// TIA Portal V18 export
FUNCTION_BLOCK "Aux_Functions"   // FB16, LAD
TITLE = Aux_Functions
{ S7_Optimized_Access := 'TRUE' }
// Written BY Kristopher Gimenez January 26,2023
// This block is used to control TD auxilarry functions
// stored: AutoNumber false, MemoryReserve 100, SetENOAutomatically false
   VAR
      PTO_Pulse { S7_SetPoint := 'True'} : TP_TIME;
      BUWOpenCLKTOffTime { S7_SetPoint := 'True'} : TP_TIME;
      BUWOpenCLKOnTime { S7_SetPoint := 'True'} : TP_TIME;
      BUWCloseHoldTOF { S7_SetPoint := 'True'} : TOF_TIME;
      MUDoneTP { S7_SetPoint := 'True'} : TP_TIME;
      BUWOpPulse { S7_SetPoint := 'True'} : TP_TIME;
      ElevCl_TON { S7_SetPoint := 'True'} : TON_TIME;
      ElevOpTime_TP { S7_SetPoint := 'True'} : TP_TIME;
      MSVOp_TON { S7_SetPoint := 'True'} : TON_TIME;
      MPRunning_TOF { S7_SetPoint := 'True'} : TOF_TIME;
      MSVCl_TON { S7_SetPoint := 'True'} : TON_TIME;
      BUWMainCl_Int { S7_SetPoint := 'True'} : Bool;
      TDModeMUTrig : Bool;
      TDModeBOTrig { ExternalAccessible := 'False'; ExternalVisible := 'False'; ExternalWritable := 'False'} : Bool;
      ElevOpOnTime : Bool;   // Bool that will be high for 8 seconds while elevator opens
      LinksDisable : Bool;   // Link Tilt Extend and Retract disabled
      ElevClDisable : Bool;   // Disable Close after output on for set time
      MSVClDisable { S7_SetPoint := 'True'} : Bool;   // MSV close disabled due to mud Pump running if high
      MSVOpDisable { S7_SetPoint := 'True'} : Bool;   // Disable after output on for set time
      ElevOpSwTrig : Bool;
      ElevCl_TON_1 { S7_SetPoint := 'True'} : TON_TIME;
      ElevCl_TON_5s { S7_SetPoint := 'True'} : TON_TIME;
   END_VAR
   // PTO_Pulse.PT := T#5s;
   VAR_TEMP   // added for the SCL form of the ladder/FBD networks
      _w1 : Bool;
      _w2 : Bool;
   END_VAR
BEGIN

REGION Network 1: PTO Pulse
   // When PTO is pressed there will be a 5 seconds pulse allowing operations.
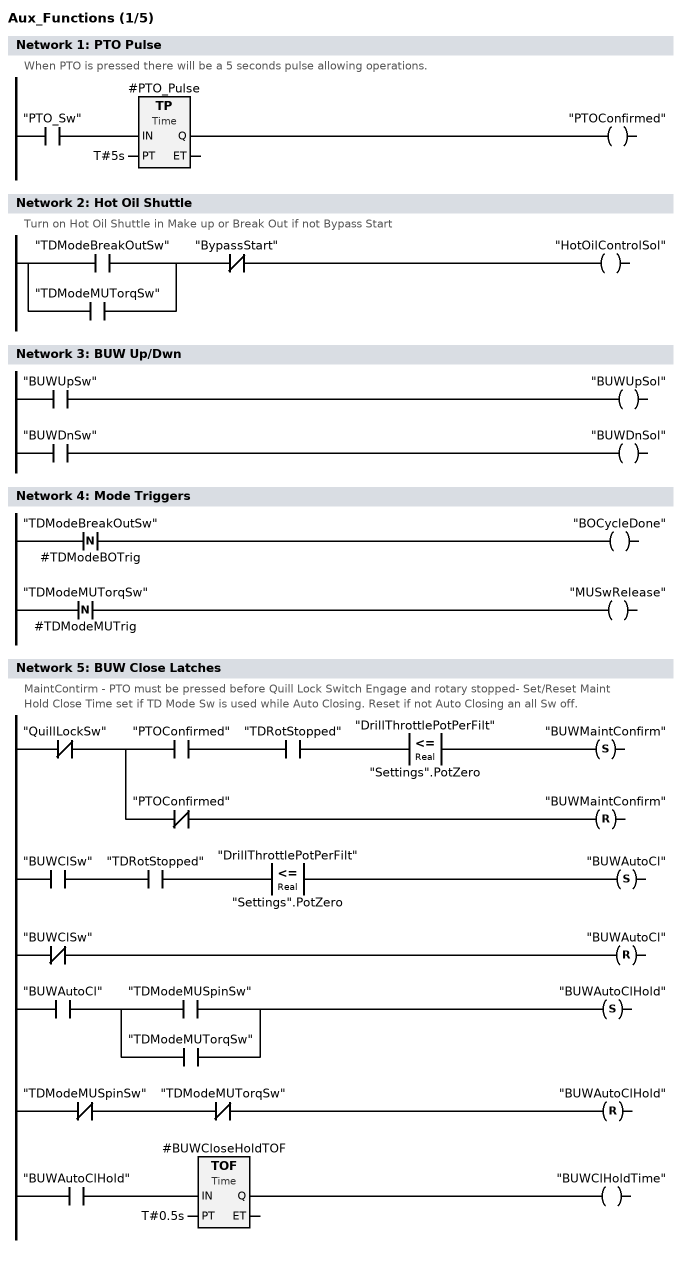
   RUNG wire#powerrail
      Contact( "PTO_Sw" )
      { S7_Templates := "time_type := Time" } #PTO_Pulse.TP(pt := T#5s, et =>)
      Coil( "PTOConfirmed" )
   END_RUNG
   // the same network as SCL:
   #PTO_Pulse(IN := "PTO_Sw", PT := T#5s);   // TP
   "PTOConfirmed" := #PTO_Pulse.Q;
END_REGION

REGION Network 2: Hot Oil Shuttle
   // Turn on Hot Oil Shuttle in Make up or Break Out if not Bypass Start
   RUNG wire#powerrail
      Contact( "TDModeBreakOutSw" )
      wire#w1
      I_Contact( "BypassStart" )
      Coil( "HotOilControlSol" )
   END_RUNG
   RUNG wire#powerrail
      Contact( "TDModeMUTorqSw" )
   END_RUNG wire#w1
   // the same network as SCL:
   "HotOilControlSol" := ("TDModeBreakOutSw" OR "TDModeMUTorqSw") AND NOT "BypassStart";
END_REGION

REGION Network 3: BUW Up/Dwn
   RUNG wire#powerrail
      Contact( "BUWUpSw" )
      Coil( "BUWUpSol" )
   END_RUNG
   RUNG wire#powerrail
      Contact( "BUWDnSw" )
      Coil( "BUWDnSol" )
   END_RUNG
   // the same network as SCL:
   "BUWUpSol" := "BUWUpSw";
   "BUWDnSol" := "BUWDnSw";
END_REGION

REGION Network 4: Mode Triggers
   RUNG wire#powerrail
      N_Contact(operand := "TDModeBreakOutSw", bit := #TDModeBOTrig)
      Coil( "BOCycleDone" )
   END_RUNG
   RUNG wire#powerrail
      N_Contact(operand := "TDModeMUTorqSw", bit := #TDModeMUTrig)
      Coil( "MUSwRelease" )
   END_RUNG
   // the same network as SCL:
   #_w1 := NOT "TDModeBreakOutSw" AND #TDModeBOTrig;   // falling edge of "TDModeBreakOutSw"
   #TDModeBOTrig := "TDModeBreakOutSw";
   "BOCycleDone" := #_w1;
   #_w2 := NOT "TDModeMUTorqSw" AND #TDModeMUTrig;   // falling edge of "TDModeMUTorqSw"
   #TDModeMUTrig := "TDModeMUTorqSw";
   "MUSwRelease" := #_w2;
END_REGION

REGION Network 5: BUW Close Latches
   // MaintContirm - PTO must be pressed before Quill Lock Switch Engage and rotary stopped- Set/Reset Maint
   // Hold Close Time set if TD Mode Sw is used while Auto Closing. Reset if not Auto Closing an all Sw off.
   RUNG wire#powerrail
      I_Contact( "QuillLockSw" )
      wire#w1
      Contact( "PTOConfirmed" )
      Contact( "TDRotStopped" )
      { S7_Templates := "SrcType := Real" } LE_Contact(in1 := "DrillThrottlePotPerFilt", in2 := "Settings".PotZero)
      S_Coil( "BUWMaintConfirm" )
   END_RUNG
   RUNG wire#w1
      I_Contact( "PTOConfirmed" )
      R_Coil( "BUWMaintConfirm" )
   END_RUNG
   RUNG wire#powerrail
      Contact( "BUWClSw" )
      Contact( "TDRotStopped" )
      { S7_Templates := "SrcType := Real" } LE_Contact(in1 := "DrillThrottlePotPerFilt", in2 := "Settings".PotZero)
      S_Coil( "BUWAutoCl" )
   END_RUNG
   RUNG wire#powerrail
      I_Contact( "BUWClSw" )
      R_Coil( "BUWAutoCl" )
   END_RUNG
   RUNG wire#powerrail
      Contact( "BUWAutoCl" )
      wire#w2
      Contact( "TDModeMUSpinSw" )
      wire#w3
      S_Coil( "BUWAutoClHold" )
   END_RUNG
   RUNG wire#w2
      Contact( "TDModeMUTorqSw" )
   END_RUNG wire#w3
   RUNG wire#powerrail
      I_Contact( "TDModeMUSpinSw" )
      I_Contact( "TDModeMUTorqSw" )
      R_Coil( "BUWAutoClHold" )
   END_RUNG
   RUNG wire#powerrail
      Contact( "BUWAutoClHold" )
      { S7_Templates := "time_type := Time" } #BUWCloseHoldTOF.TOF(pt := T#0.5s, et =>)
      Coil( "BUWClHoldTime" )
   END_RUNG
   // the same network as SCL:
   IF NOT "QuillLockSw" AND "PTOConfirmed" AND "TDRotStopped" AND ("DrillThrottlePotPerFilt" <= "Settings".PotZero) THEN
       "BUWMaintConfirm" := TRUE;
   END_IF;
   IF NOT "QuillLockSw" AND NOT "PTOConfirmed" THEN "BUWMaintConfirm" := FALSE; END_IF;
   IF "BUWClSw" AND "TDRotStopped" AND ("DrillThrottlePotPerFilt" <= "Settings".PotZero) THEN
       "BUWAutoCl" := TRUE;
   END_IF;
   IF NOT "BUWClSw" THEN "BUWAutoCl" := FALSE; END_IF;
   IF "BUWAutoCl" AND ("TDModeMUSpinSw" OR "TDModeMUTorqSw") THEN "BUWAutoClHold" := TRUE; END_IF;
   IF NOT "TDModeMUSpinSw" AND NOT "TDModeMUTorqSw" THEN "BUWAutoClHold" := FALSE; END_IF;
   #BUWCloseHoldTOF(IN := "BUWAutoClHold", PT := T#0.5s);   // TOF
   "BUWClHoldTime" := #BUWCloseHoldTOF.Q;
END_REGION

REGION Network 6: BUW Auto Open Latch
   // Auto open if Break out finished or Makeup sw released
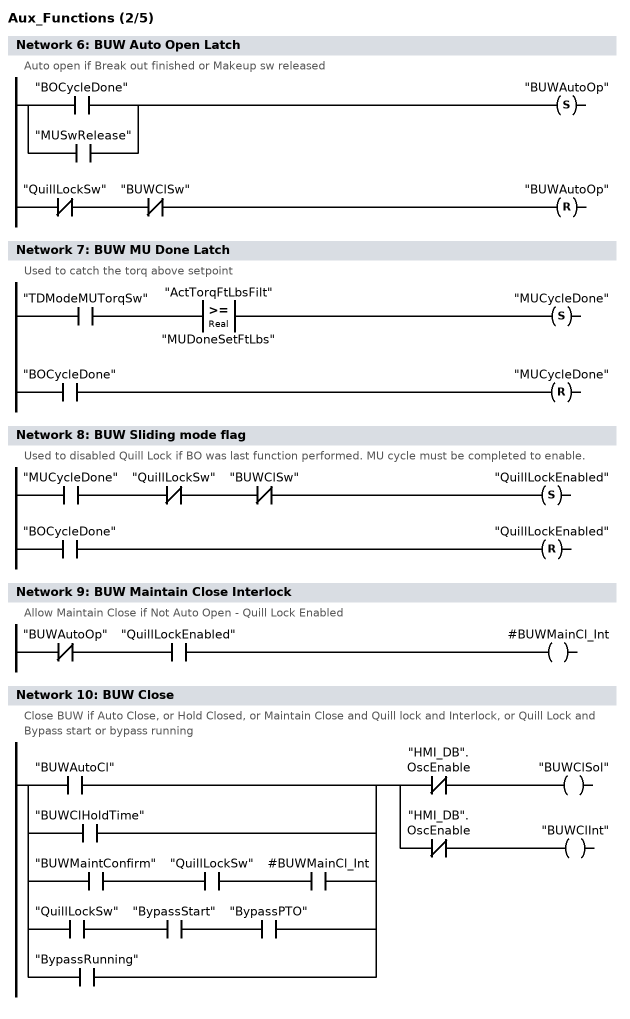
   RUNG wire#powerrail
      Contact( "BOCycleDone" )
      wire#w1
      S_Coil( "BUWAutoOp" )
   END_RUNG
   RUNG wire#powerrail
      Contact( "MUSwRelease" )
   END_RUNG wire#w1
   RUNG wire#powerrail
      I_Contact( "QuillLockSw" )
      I_Contact( "BUWClSw" )
      R_Coil( "BUWAutoOp" )
   END_RUNG
   // the same network as SCL:
   IF "BOCycleDone" OR "MUSwRelease" THEN "BUWAutoOp" := TRUE; END_IF;
   IF NOT "QuillLockSw" AND NOT "BUWClSw" THEN "BUWAutoOp" := FALSE; END_IF;
END_REGION

REGION Network 7: BUW MU Done Latch
   // Used to catch the torq above setpoint
   RUNG wire#powerrail
      Contact( "TDModeMUTorqSw" )
      { S7_Templates := "SrcType := Real" } GE_Contact(in1 := "ActTorqFtLbsFilt", in2 := "MUDoneSetFtLbs")
      S_Coil( "MUCycleDone" )
   END_RUNG
   RUNG wire#powerrail
      Contact( "BOCycleDone" )
      R_Coil( "MUCycleDone" )
   END_RUNG
   // the same network as SCL:
   IF "TDModeMUTorqSw" AND ("ActTorqFtLbsFilt" >= "MUDoneSetFtLbs") THEN "MUCycleDone" := TRUE; END_IF;
   IF "BOCycleDone" THEN "MUCycleDone" := FALSE; END_IF;
END_REGION

REGION Network 8: BUW Sliding mode flag
   // Used to disabled Quill Lock if BO was last function performed. MU cycle must be completed to enable.
   RUNG wire#powerrail
      Contact( "MUCycleDone" )
      I_Contact( "QuillLockSw" )
      I_Contact( "BUWClSw" )
      S_Coil( "QuillLockEnabled" )
   END_RUNG
   RUNG wire#powerrail
      Contact( "BOCycleDone" )
      R_Coil( "QuillLockEnabled" )
   END_RUNG
   // the same network as SCL:
   IF "MUCycleDone" AND NOT "QuillLockSw" AND NOT "BUWClSw" THEN "QuillLockEnabled" := TRUE; END_IF;
   IF "BOCycleDone" THEN "QuillLockEnabled" := FALSE; END_IF;
END_REGION

REGION Network 9: BUW Maintain Close Interlock
   // Allow Maintain Close if Not Auto Open - Quill Lock Enabled
   RUNG wire#powerrail
      I_Contact( "BUWAutoOp" )
      Contact( "QuillLockEnabled" )
      Coil( #BUWMainCl_Int )
   END_RUNG
   // the same network as SCL:
   #BUWMainCl_Int := NOT "BUWAutoOp" AND "QuillLockEnabled";
END_REGION

REGION Network 10: BUW Close
   // Close BUW if Auto Close, or Hold Closed, or Maintain Close and Quill lock and Interlock, or Quill Lock and Bypass start or bypass running
   RUNG wire#powerrail
      Contact( "BUWAutoCl" )
      wire#w1
      I_Contact( "HMI_DB".OscEnable )
      Coil( "BUWClSol" )
   END_RUNG
   RUNG wire#powerrail
      Contact( "BUWClHoldTime" )
   END_RUNG wire#w1
   RUNG wire#powerrail
      Contact( "BUWMaintConfirm" )
      Contact( "QuillLockSw" )
      Contact( #BUWMainCl_Int )
   END_RUNG wire#w1
   RUNG wire#powerrail
      Contact( "QuillLockSw" )
      Contact( "BypassStart" )
      Contact( "BypassPTO" )
   END_RUNG wire#w1
   RUNG wire#powerrail
      Contact( "BypassRunning" )
   END_RUNG wire#w1
   RUNG wire#w1
      I_Contact( "HMI_DB".OscEnable )
      Coil( "BUWClInt" )
   END_RUNG
   // the same network as SCL:
   #_w1 := "BUWAutoCl" OR "BUWClHoldTime" OR ("BUWMaintConfirm" AND "QuillLockSw" AND #BUWMainCl_Int) OR ("QuillLockSw" AND "BypassStart" AND "BypassPTO") OR "BypassRunning";
   "BUWClSol" := #_w1 AND NOT "HMI_DB".OscEnable;
   "BUWClInt" := #_w1 AND NOT "HMI_DB".OscEnable;
END_REGION

REGION Network 11: BUW Open Clock
   // Clock is on for 5 seconds a minute when Not BUW Cl, not Quill lock, not gripper close and throttle>zero
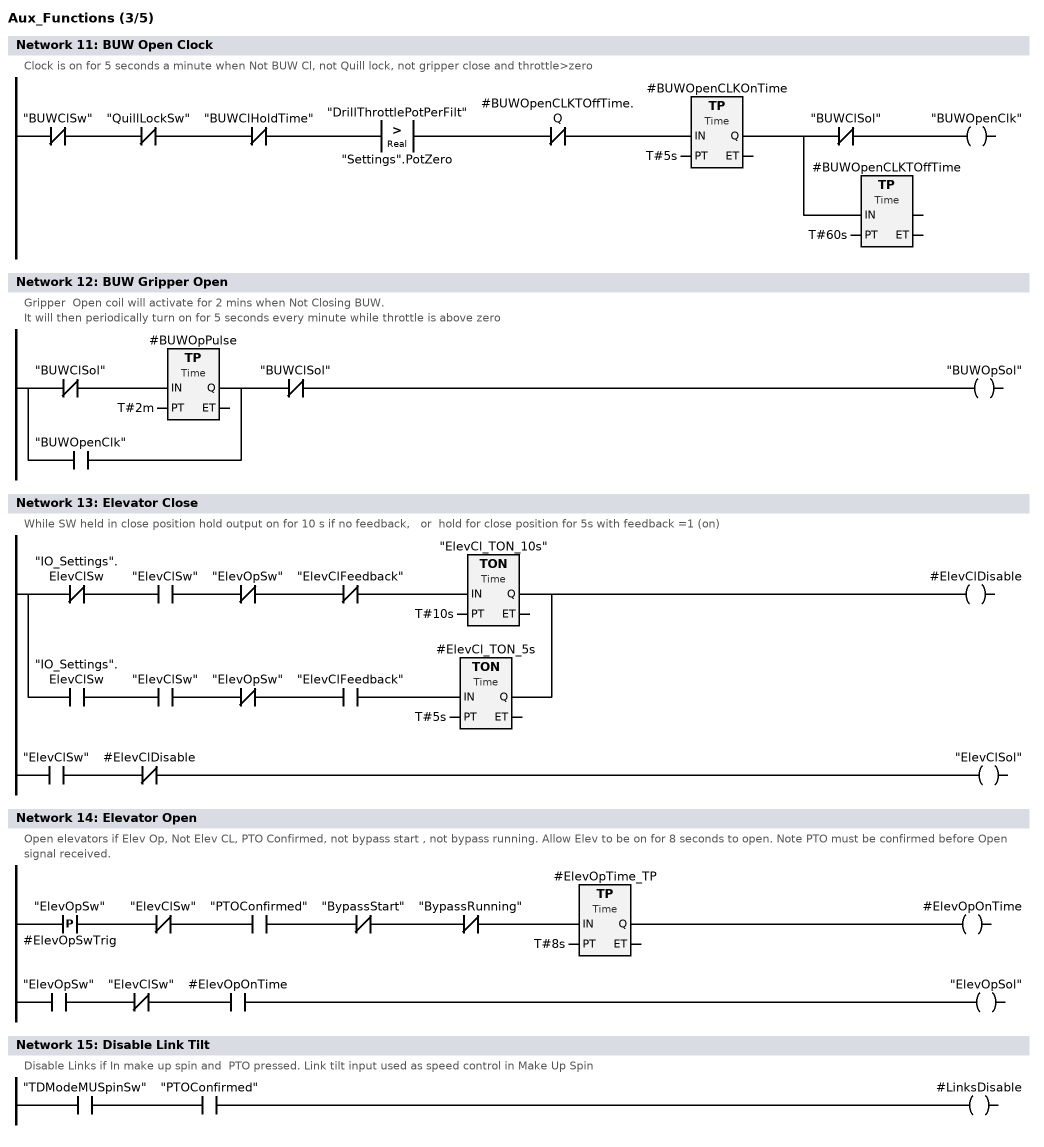
   RUNG wire#powerrail
      I_Contact( "BUWClSw" )
      I_Contact( "QuillLockSw" )
      I_Contact( "BUWClHoldTime" )
      { S7_Templates := "SrcType := Real" } GT_Contact(in1 := "DrillThrottlePotPerFilt", in2 := "Settings".PotZero)
      I_Contact( #BUWOpenCLKTOffTime.Q )
      { S7_Templates := "time_type := Time" } #BUWOpenCLKOnTime.TP(pt := T#5s, et =>)
      wire#w1
      I_Contact( "BUWClSol" )
      Coil( "BUWOpenClk" )
   END_RUNG
   RUNG wire#w1
      { S7_Templates := "time_type := Time" } #BUWOpenCLKTOffTime.TP(pt := T#60s, et =>)
   END_RUNG
   // the same network as SCL:
   #BUWOpenCLKOnTime(IN := NOT "BUWClSw" AND NOT "QuillLockSw" AND NOT "BUWClHoldTime" AND ("DrillThrottlePotPerFilt" > "Settings".PotZero) AND NOT #BUWOpenCLKTOffTime.Q,   // TP
                     PT := T#5s);
   "BUWOpenClk" := #BUWOpenCLKOnTime.Q AND NOT "BUWClSol";
   #BUWOpenCLKTOffTime(IN := #BUWOpenCLKOnTime.Q, PT := T#60s);   // TP
END_REGION

REGION Network 12: BUW Gripper Open
   // Gripper  Open coil will activate for 2 mins when Not Closing BUW. 
   // It will then periodically turn on for 5 seconds every minute while throttle is above zero
   RUNG wire#powerrail
      I_Contact( "BUWClSol" )
      { S7_Templates := "time_type := Time" } #BUWOpPulse.TP(pt := T#2m, et =>)
      wire#w1
      I_Contact( "BUWClSol" )
      Coil( "BUWOpSol" )
   END_RUNG
   RUNG wire#powerrail
      Contact( "BUWOpenClk" )
   END_RUNG wire#w1
   // the same network as SCL:
   #BUWOpPulse(IN := NOT "BUWClSol", PT := T#2m);   // TP
   "BUWOpSol" := (#BUWOpPulse.Q OR "BUWOpenClk") AND NOT "BUWClSol";
END_REGION

REGION Network 13: Elevator Close
   // While SW held in close position hold output on for 10 s if no feedback,   or  hold for close position for 5s with feedback =1 (on)
   RUNG wire#powerrail
      I_Contact( "IO_Settings".ElevClSw )
      Contact( "ElevClSw" )
      I_Contact( "ElevOpSw" )
      I_Contact( "ElevClFeedback" )
      { S7_Templates := "time_type := Time" } "ElevCl_TON_10s".TON(pt := T#10s, et =>)
      wire#w1
      Coil( #ElevClDisable )
   END_RUNG
   RUNG wire#powerrail
      Contact( "IO_Settings".ElevClSw )
      Contact( "ElevClSw" )
      I_Contact( "ElevOpSw" )
      Contact( "ElevClFeedback" )
      { S7_Templates := "time_type := Time" } #ElevCl_TON_5s.TON(pt := T#5s, et =>)
   END_RUNG wire#w1
   RUNG wire#powerrail
      Contact( "ElevClSw" )
      I_Contact( #ElevClDisable )
      Coil( "ElevClSol" )
   END_RUNG
   // the same network as SCL:
   "ElevCl_TON_10s".TON(IN := NOT "IO_Settings".ElevClSw AND "ElevClSw" AND NOT "ElevOpSw" AND NOT "ElevClFeedback",
                        PT := T#10s);
   #ElevCl_TON_5s(IN := "IO_Settings".ElevClSw AND "ElevClSw" AND NOT "ElevOpSw" AND "ElevClFeedback",   // TON
                  PT := T#5s);
   #ElevClDisable := "ElevCl_TON_10s".Q OR #ElevCl_TON_5s.Q;
   "ElevClSol" := "ElevClSw" AND NOT #ElevClDisable;
END_REGION

REGION Network 14: Elevator Open
   // Open elevators if Elev Op, Not Elev CL, PTO Confirmed, not bypass start , not bypass running. Allow Elev to be on for 8 seconds to open. Note PTO must be confirmed before Open signal received.
   RUNG wire#powerrail
      P_Contact(operand := "ElevOpSw", bit := #ElevOpSwTrig)
      I_Contact( "ElevClSw" )
      Contact( "PTOConfirmed" )
      I_Contact( "BypassStart" )
      I_Contact( "BypassRunning" )
      { S7_Templates := "time_type := Time" } #ElevOpTime_TP.TP(pt := T#8s, et =>)
      Coil( #ElevOpOnTime )
   END_RUNG
   RUNG wire#powerrail
      Contact( "ElevOpSw" )
      I_Contact( "ElevClSw" )
      Contact( #ElevOpOnTime )
      Coil( "ElevOpSol" )
   END_RUNG
   // the same network as SCL:
   #_w1 := "ElevOpSw" AND NOT #ElevOpSwTrig;   // rising edge of "ElevOpSw"
   #ElevOpSwTrig := "ElevOpSw";
   #ElevOpTime_TP(IN := #_w1 AND NOT "ElevClSw" AND "PTOConfirmed" AND NOT "BypassStart" AND NOT "BypassRunning",   // TP
                  PT := T#8s);
   #ElevOpOnTime := #ElevOpTime_TP.Q;
   "ElevOpSol" := "ElevOpSw" AND NOT "ElevClSw" AND #ElevOpOnTime;
END_REGION

REGION Network 15: Disable Link Tilt
   // Disable Links if In make up spin and  PTO pressed. Link tilt input used as speed control in Make Up Spin
   RUNG wire#powerrail
      Contact( "TDModeMUSpinSw" )
      Contact( "PTOConfirmed" )
      Coil( #LinksDisable )
   END_RUNG
   // the same network as SCL:
   #LinksDisable := "TDModeMUSpinSw" AND "PTOConfirmed";
END_REGION

REGION Network 16: Link Tilts
   // No Ext/Ret if links disabled
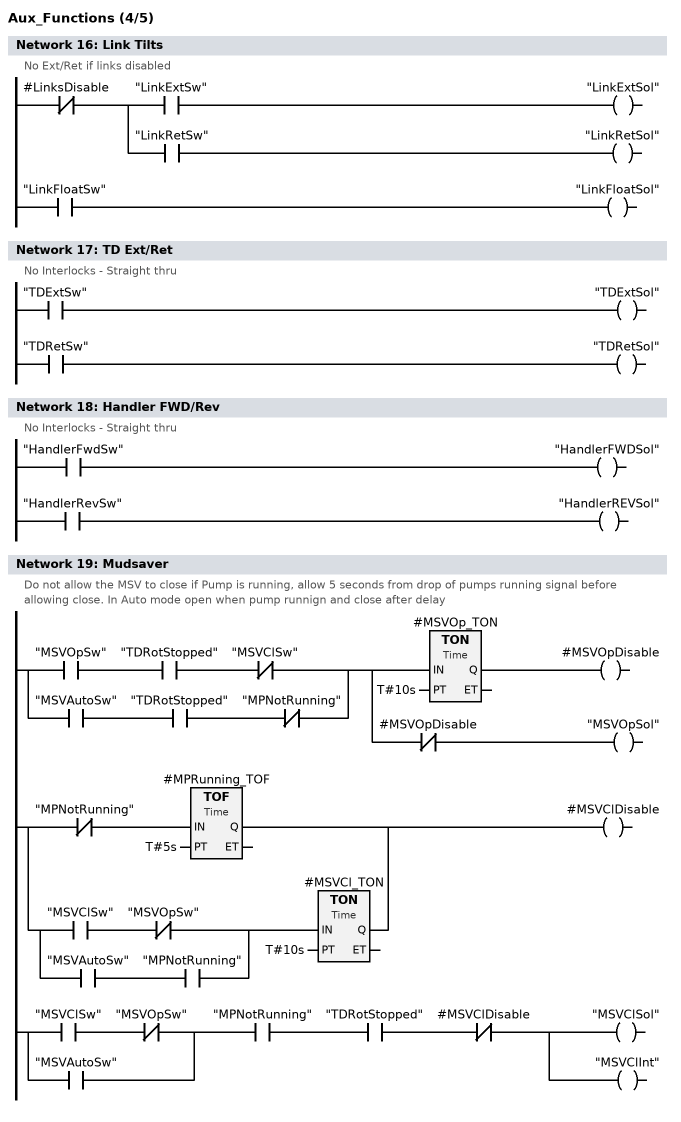
   RUNG wire#powerrail
      I_Contact( #LinksDisable )
      wire#w1
      Contact( "LinkExtSw" )
      Coil( "LinkExtSol" )
   END_RUNG
   RUNG wire#w1
      Contact( "LinkRetSw" )
      Coil( "LinkRetSol" )
   END_RUNG
   RUNG wire#powerrail
      Contact( "LinkFloatSw" )
      Coil( "LinkFloatSol" )
   END_RUNG
   // the same network as SCL:
   "LinkExtSol" := NOT #LinksDisable AND "LinkExtSw";
   "LinkRetSol" := NOT #LinksDisable AND "LinkRetSw";
   "LinkFloatSol" := "LinkFloatSw";
END_REGION

REGION Network 17: TD Ext/Ret
   // No Interlocks - Straight thru
   RUNG wire#powerrail
      Contact( "TDExtSw" )
      Coil( "TDExtSol" )
   END_RUNG
   RUNG wire#powerrail
      Contact( "TDRetSw" )
      Coil( "TDRetSol" )
   END_RUNG
   // the same network as SCL:
   "TDExtSol" := "TDExtSw";
   "TDRetSol" := "TDRetSw";
END_REGION

REGION Network 18: Handler FWD/Rev
   // No Interlocks - Straight thru
   RUNG wire#powerrail
      Contact( "HandlerFwdSw" )
      Coil( "HandlerFWDSol" )
   END_RUNG
   RUNG wire#powerrail
      Contact( "HandlerRevSw" )
      Coil( "HandlerREVSol" )
   END_RUNG
   // the same network as SCL:
   "HandlerFWDSol" := "HandlerFwdSw";
   "HandlerREVSol" := "HandlerRevSw";
END_REGION

REGION Network 19: Mudsaver
   // Do not allow the MSV to close if Pump is running, allow 5 seconds from drop of pumps running signal before allowing close. In Auto mode open when pump runnign and close after delay
   RUNG wire#powerrail
      Contact( "MSVOpSw" )
      Contact( "TDRotStopped" )
      I_Contact( "MSVClSw" )
      wire#w1
      { S7_Templates := "time_type := Time" } #MSVOp_TON.TON(pt := T#10s, et =>)
      Coil( #MSVOpDisable )
   END_RUNG
   RUNG wire#powerrail
      Contact( "MSVAutoSw" )
      Contact( "TDRotStopped" )
      I_Contact( "MPNotRunning" )
   END_RUNG wire#w1
   RUNG wire#w1
      I_Contact( #MSVOpDisable )
      Coil( "MSVOpSol" )
   END_RUNG
   RUNG wire#powerrail
      I_Contact( "MPNotRunning" )
      { S7_Templates := "time_type := Time" } #MPRunning_TOF.TOF(pt := T#5s, et =>)
      wire#w2
      Coil( #MSVClDisable )
   END_RUNG
   RUNG wire#powerrail
      Contact( "MSVClSw" )
      I_Contact( "MSVOpSw" )
      wire#w3
      { S7_Templates := "time_type := Time" } #MSVCl_TON.TON(pt := T#10s, et =>)
   END_RUNG wire#w2
   RUNG wire#powerrail
      Contact( "MSVAutoSw" )
      Contact( "MPNotRunning" )
   END_RUNG wire#w3
   RUNG wire#powerrail
      Contact( "MSVClSw" )
      I_Contact( "MSVOpSw" )
      wire#w4
      Contact( "MPNotRunning" )
      Contact( "TDRotStopped" )
      I_Contact( #MSVClDisable )
      wire#w5
      Coil( "MSVClSol" )
   END_RUNG
   RUNG wire#powerrail
      Contact( "MSVAutoSw" )
   END_RUNG wire#w4
   RUNG wire#w5
      Coil( "MSVClInt" )
   END_RUNG
   // the same network as SCL:
   #_w1 := ("MSVOpSw" AND "TDRotStopped" AND NOT "MSVClSw") OR ("MSVAutoSw" AND "TDRotStopped" AND NOT "MPNotRunning");
   #MSVOp_TON(IN := #_w1, PT := T#10s);   // TON
   #MSVOpDisable := #MSVOp_TON.Q;
   "MSVOpSol" := #_w1 AND NOT #MSVOpDisable;
   #MPRunning_TOF(IN := NOT "MPNotRunning", PT := T#5s);   // TOF
   #MSVCl_TON(IN := ("MSVClSw" AND NOT "MSVOpSw") OR ("MSVAutoSw" AND "MPNotRunning"), PT := T#10s);   // TON
   #MSVClDisable := #MPRunning_TOF.Q OR #MSVCl_TON.Q;
   "MSVClSol" := (("MSVClSw" AND NOT "MSVOpSw") OR "MSVAutoSw") AND "MPNotRunning" AND "TDRotStopped" AND NOT #MSVClDisable;
   "MSVClInt" := "MSVClSol";
END_REGION

REGION Network 20: Unloader
   // Unloader is valve is on if Drill throttle greater than zero and no Auxiliary functions are being used
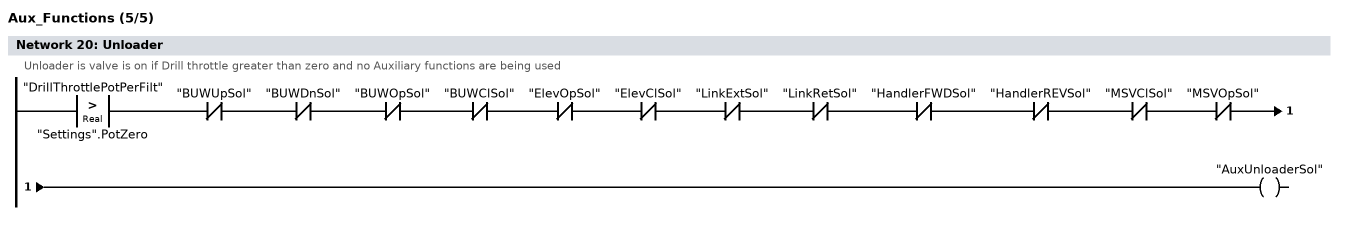
   RUNG wire#powerrail
      { S7_Templates := "SrcType := Real" } GT_Contact(in1 := "DrillThrottlePotPerFilt", in2 := "Settings".PotZero)
      I_Contact( "BUWUpSol" )
      I_Contact( "BUWDnSol" )
      I_Contact( "BUWOpSol" )
      I_Contact( "BUWClSol" )
      I_Contact( "ElevOpSol" )
      I_Contact( "ElevClSol" )
      I_Contact( "LinkExtSol" )
      I_Contact( "LinkRetSol" )
      I_Contact( "HandlerFWDSol" )
      I_Contact( "HandlerREVSol" )
      I_Contact( "MSVClSol" )
      I_Contact( "MSVOpSol" )
      Coil( "AuxUnloaderSol" )
   END_RUNG
   // the same network as SCL:
   "AuxUnloaderSol" := ("DrillThrottlePotPerFilt" > "Settings".PotZero) AND NOT "BUWUpSol" AND NOT "BUWDnSol" AND NOT "BUWOpSol" AND NOT "BUWClSol" AND NOT "ElevOpSol" AND NOT "ElevClSol" AND NOT "LinkExtSol" AND NOT "LinkRetSol" AND NOT "HandlerFWDSol" AND NOT "HandlerREVSol" AND NOT "MSVClSol" AND NOT "MSVOpSol";
END_REGION
END_FUNCTION_BLOCK
